// TIA Portal project "2022.11.20_三轴机械臂仿真" (V17)
// Vorlageprojekt für das Buch mit Zielsystem S7-1200

(* hardware
DEVICE "S7-1200-Station_1"  S7-1200 Station
   slot 0: "Baugruppenträger_0"  Rack  V1.0
   slot 1: "PLC_1"  CPU 1214C DC/DC/DC  6ES7 214-1AG40-0XB0  V4.5
*)

// ===== PLC "PLC_1"  CPU 1214C DC/DC/DC =====

VAR_GLOBAL   // PLC tag table "Standard-Variablentabelle"
   "传送带1" AT %A0.0 : Bool;
   "感应器1" AT %E0.0 : Bool;
   "感应器2" AT %E0.1 : Bool;
   "启动" AT %M10.0 : Bool;
   "暂停按钮" AT %I0.2 : Bool;
   "吸物" AT %Q0.3 : Bool;
   "传送带2" AT %Q0.1 : Bool;
   "传送带3" AT %Q0.2 : Bool;
   "上升沿暂存位1" AT %M100.0 : Bool;
   "传送带1输出" AT %M20.0 : Bool;
   "完成" AT %M30.7 : Bool;
   "上升沿暂存位2" AT %M100.1 : Bool;
   "碰上感应1" AT %M30.0 : Bool;
   "传送带3输出" AT %M20.2 : Bool;
   "上升沿暂存位3" AT %M100.2 : Bool;
   "开始拿物" AT %M30.2 : Bool;
   "循环" AT %M30.6 : Bool;
   "碰上感应2" AT %M30.1 : Bool;
   "完成拿物" AT %M30.3 : Bool;
   "X输出" AT %QD30 : Real;
   "Y输出" AT %QD34 : Real;
   "X位置" AT %ID30 : DWord;
   "Y位置" AT %ID34 : DWord;
   "Z输出" AT %QD38 : Real;
   "Z位置" AT %ID38 : DWord;
   "吸物输出" AT %M20.3 : Bool;
   "上升沿暂存位4" AT %M100.3 : Bool;
   "物体个数" AT %MD50 : DWord;
   "X设置输出" AT %MD54 : DWord;
   "Y设置输出" AT %MD58 : DWord;
   "上升沿暂存位5" AT %M100.4 : Bool;
   "X位置(1)" AT %MD62 : Real;
   "Y位置(1)" AT %MD66 : Real;
   "Tag_2" AT %MD34 : DWord;
   "下降" AT %M30.4 : Bool;
   "上升沿暂存位" AT %M100.5 : Bool;
   "Z设置输出" AT %MD70 : Real;
   "Z位置(1)" AT %MD74 : Real;
   "Z位置(2)" AT %MD38 : DWord;
   "上升" AT %M30.5 : Bool;
   "上升沿暂存位(1)" AT %M100.6 : Bool;
   "停止" AT %M10.1 : Bool;
   "Tag_3" AT %M20.1 : Bool;
END_VAR

DATA_BLOCK "拿物_DB"   // DB1
{ S7_Optimized_Access := 'TRUE' }
VERSION : 0.1
// stored: InstanceOfName 拿物
"拿物"
BEGIN
END_DATA_BLOCK

DATA_BLOCK "放物_DB"   // DB10
{ S7_Optimized_Access := 'TRUE' }
VERSION : 0.1
// stored: InstanceOfName 放物
"放物"
BEGIN
END_DATA_BLOCK

DATA_BLOCK "输出_DB"   // DB11
{ S7_Optimized_Access := 'TRUE' }
VERSION : 0.1
// stored: InstanceOfName 输出
"输出"
BEGIN
END_DATA_BLOCK

// folder: System blocks/Program resources

DATA_BLOCK "计数器1"   // DB2
{ S7_Optimized_Access := 'TRUE' }
AUTHOR : Simatic
FAMILY : IEC
NAME : CNTR
VERSION : 1.0
// stored: InstanceOfName IEC_COUNTER
"IEC_COUNTER"
BEGIN
END_DATA_BLOCK

DATA_BLOCK "计数器2"   // DB4
{ S7_Optimized_Access := 'TRUE' }
AUTHOR : Simatic
FAMILY : IEC
NAME : CNTR
VERSION : 1.0
// stored: InstanceOfName IEC_COUNTER
"IEC_COUNTER"
BEGIN
END_DATA_BLOCK

DATA_BLOCK "计时器1"   // DB5
{ S7_Optimized_Access := 'TRUE' }
AUTHOR : Simatic
FAMILY : IEC
NAME : IEC_TMR
VERSION : 1.0
// stored: InstanceOfName IEC_TIMER
"IEC_TIMER"
BEGIN
END_DATA_BLOCK

DATA_BLOCK "计数器3"   // DB6
{ S7_Optimized_Access := 'TRUE' }
AUTHOR : Simatic
FAMILY : IEC
NAME : CNTR
VERSION : 1.0
// stored: InstanceOfName IEC_COUNTER
"IEC_COUNTER"
BEGIN
END_DATA_BLOCK

DATA_BLOCK "计时器2"   // DB7
{ S7_Optimized_Access := 'TRUE' }
AUTHOR : Simatic
FAMILY : IEC
NAME : IEC_TMR
VERSION : 1.0
// stored: InstanceOfName IEC_TIMER
"IEC_TIMER"
BEGIN
END_DATA_BLOCK

DATA_BLOCK "计时2"   // DB8
{ S7_Optimized_Access := 'TRUE' }
AUTHOR : Simatic
FAMILY : IEC
NAME : IEC_TMR
VERSION : 1.0
// stored: InstanceOfName IEC_TIMER
"IEC_TIMER"
BEGIN
END_DATA_BLOCK

DATA_BLOCK "计时1"   // DB9
{ S7_Optimized_Access := 'TRUE' }
AUTHOR : Simatic
FAMILY : IEC
NAME : IEC_TMR
VERSION : 1.0
// stored: InstanceOfName IEC_TIMER
"IEC_TIMER"
BEGIN
END_DATA_BLOCK

// folder: (top level)

FUNCTION_BLOCK "拿物"   // FB1, LAD
{ S7_Optimized_Access := 'TRUE' }
VERSION : 0.1
   VAR_TEMP   // added for the SCL form of the ladder/FBD networks
      _w1 : Bool;
   END_VAR
BEGIN

REGION Network 1: 2个感应碰上后开始拿物
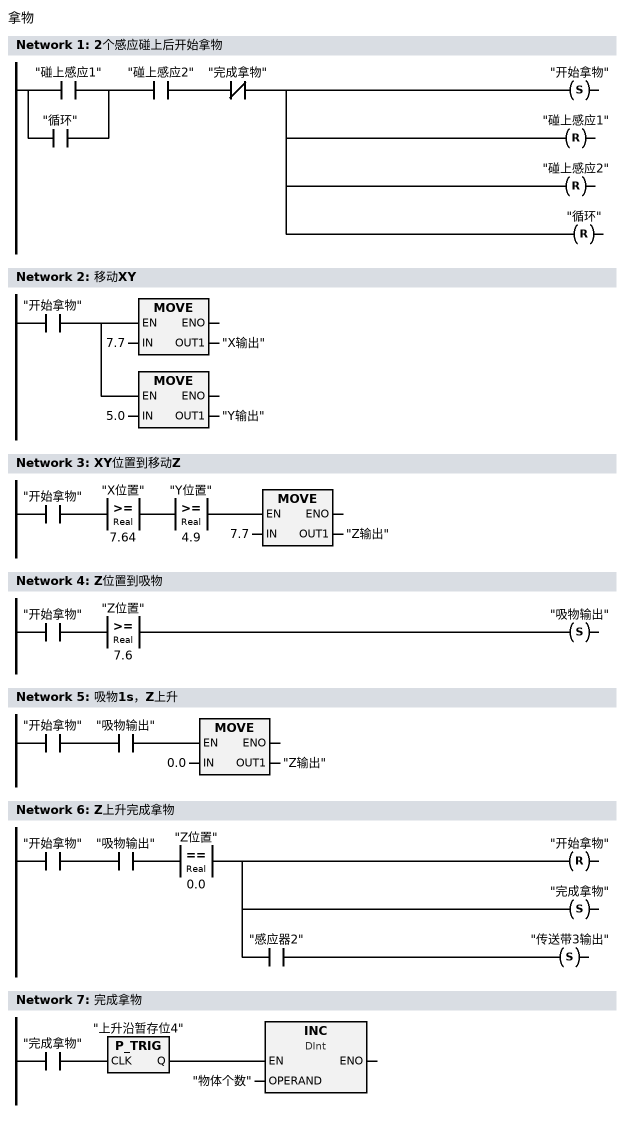
   RUNG wire#powerrail
      Contact( "碰上感应1" )
      wire#w1
      Contact( "碰上感应2" )
      I_Contact( "完成拿物" )
      wire#w2
      S_Coil( "开始拿物" )
   END_RUNG
   RUNG wire#powerrail
      Contact( "循环" )
   END_RUNG wire#w1
   RUNG wire#w2
      R_Coil( "碰上感应1" )
   END_RUNG
   RUNG wire#w2
      R_Coil( "碰上感应2" )
   END_RUNG
   RUNG wire#w2
      R_Coil( "循环" )
   END_RUNG
   // the same network as SCL:
   IF ("碰上感应1" OR "循环") AND "碰上感应2" AND NOT "完成拿物" THEN "开始拿物" := TRUE; END_IF;
   #_w1 := ("碰上感应1" OR "循环") AND "碰上感应2" AND NOT "完成拿物";
   IF #_w1 THEN
       "碰上感应1" := FALSE;
       "碰上感应2" := FALSE;
       "循环" := FALSE;
   END_IF;
END_REGION

REGION Network 2: 移动XY
   RUNG wire#powerrail
      Contact( "开始拿物" )
      wire#w1
      Move(in := 7.7, out1 => "X输出")
   END_RUNG
   RUNG wire#w1
      Move(in := 5.0, out1 => "Y输出")
   END_RUNG
   // the same network as SCL:
   IF "开始拿物" THEN
       "X输出" := 7.7;
       "Y输出" := 5.0;
   END_IF;
END_REGION

REGION Network 3: XY位置到移动Z
   RUNG wire#powerrail
      Contact( "开始拿物" )
      { S7_Templates := "SrcType := Real" } GE_Contact(in1 := "X位置", in2 := 7.64)
      { S7_Templates := "SrcType := Real" } GE_Contact(in1 := "Y位置", in2 := 4.9)
      Move(in := 7.7, out1 => "Z输出")
   END_RUNG
   // the same network as SCL:
   IF "开始拿物" AND ("X位置" >= 7.64) AND ("Y位置" >= 4.9) THEN "Z输出" := 7.7; END_IF;
END_REGION

REGION Network 4: Z位置到吸物
   RUNG wire#powerrail
      Contact( "开始拿物" )
      { S7_Templates := "SrcType := Real" } GE_Contact(in1 := "Z位置", in2 := 7.6)
      S_Coil( "吸物输出" )
   END_RUNG
   // the same network as SCL:
   IF "开始拿物" AND ("Z位置" >= 7.6) THEN "吸物输出" := TRUE; END_IF;
END_REGION

REGION Network 5: 吸物1s，Z上升
   RUNG wire#powerrail
      Contact( "开始拿物" )
      Contact( "吸物输出" )
      Move(in := 0.0, out1 => "Z输出")
   END_RUNG
   // the same network as SCL:
   IF "开始拿物" AND "吸物输出" THEN "Z输出" := 0.0; END_IF;
END_REGION

REGION Network 6: Z上升完成拿物
   RUNG wire#powerrail
      Contact( "开始拿物" )
      Contact( "吸物输出" )
      { S7_Templates := "SrcType := Real" } EQ_Contact(in1 := "Z位置", in2 := 0.0)
      wire#w1
      R_Coil( "开始拿物" )
   END_RUNG
   RUNG wire#w1
      S_Coil( "完成拿物" )
   END_RUNG
   RUNG wire#w1
      Contact( "感应器2" )
      S_Coil( "传送带3输出" )
   END_RUNG
   // the same network as SCL:
   #_w1 := "开始拿物" AND "吸物输出" AND ("Z位置" = 0.0);
   IF #_w1 THEN
       "开始拿物" := FALSE;
       "完成拿物" := TRUE;
   END_IF;
   IF #_w1 AND "感应器2" THEN "传送带3输出" := TRUE; END_IF;
END_REGION

REGION Network 7: 完成拿物
   RUNG wire#powerrail
      Contact( "完成拿物" )
      P_Trig( "上升沿暂存位4" )
      { S7_Templates := "DestType := DInt" } Inc( "物体个数" )
   END_RUNG
   // the same network as SCL:
   #_w1 := "完成拿物" AND NOT "上升沿暂存位4";   // rising edge
   "上升沿暂存位4" := "完成拿物";
   IF #_w1 THEN "物体个数" := "物体个数" + 1; END_IF;
END_REGION
END_FUNCTION_BLOCK

FUNCTION_BLOCK "输出"   // FB2, LAD
{ S7_Optimized_Access := 'TRUE' }
VERSION : 0.1
BEGIN

REGION Network 1
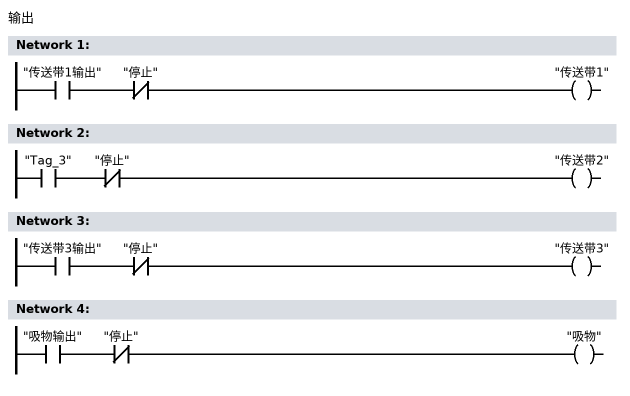
   RUNG wire#powerrail
      Contact( "传送带1输出" )
      I_Contact( "停止" )
      Coil( "传送带1" )
   END_RUNG
   // the same network as SCL:
   "传送带1" := "传送带1输出" AND NOT "停止";
END_REGION

REGION Network 2
   RUNG wire#powerrail
      Contact( "Tag_3" )
      I_Contact( "停止" )
      Coil( "传送带2" )
   END_RUNG
   // the same network as SCL:
   "传送带2" := "Tag_3" AND NOT "停止";
END_REGION

REGION Network 3
   RUNG wire#powerrail
      Contact( "传送带3输出" )
      I_Contact( "停止" )
      Coil( "传送带3" )
   END_RUNG
   // the same network as SCL:
   "传送带3" := "传送带3输出" AND NOT "停止";
END_REGION

REGION Network 4
   RUNG wire#powerrail
      Contact( "吸物输出" )
      I_Contact( "停止" )
      Coil( "吸物" )
   END_RUNG
   // the same network as SCL:
   "吸物" := "吸物输出" AND NOT "停止";
END_REGION
END_FUNCTION_BLOCK

FUNCTION_BLOCK "放物"   // FB3, LAD
{ S7_Optimized_Access := 'TRUE' }
VERSION : 0.1
   VAR_TEMP   // added for the SCL form of the ladder/FBD networks
      _w1 : Bool;
      _w2 : Bool;
   END_VAR
BEGIN

REGION Network 1: Y计数
   // 1. X: 2.3    Y:8.1   2.  X: 4.2   Y:8.0
   // 3. X: 2.3    Y:6.1   4.  X: 4.2   Y:6.0
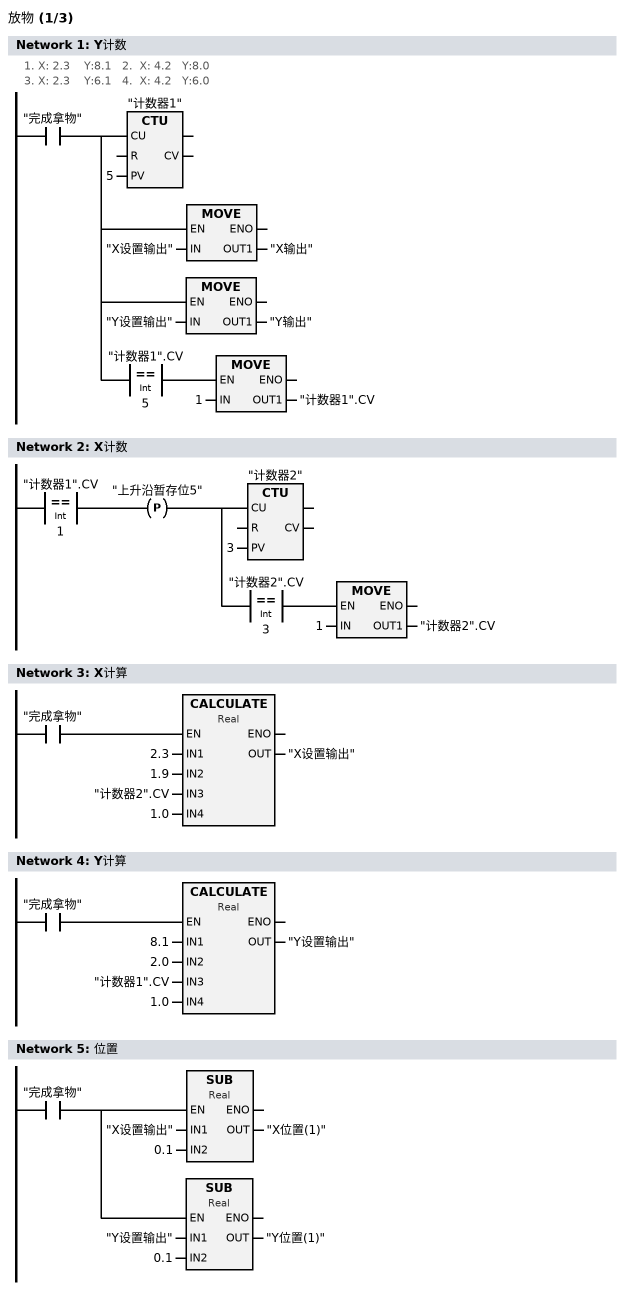
   "计数器1".CTU(CU := "完成拿物", PV := 5);
   IF "完成拿物" THEN
       "X输出" := "X设置输出";
       "Y输出" := "Y设置输出";
   END_IF;
   IF "完成拿物" AND ("计数器1".CV = 5) THEN "计数器1".CV := 1; END_IF;
END_REGION

REGION Network 2: X计数
   #_w1 := "计数器1".CV = 1;
   #_w2 := #_w1 AND NOT "上升沿暂存位5";   // rising edge
   "上升沿暂存位5" := #_w1;
   "计数器2".CTU(CU := #_w2, PV := 3);
   IF #_w2 AND ("计数器2".CV = 3) THEN "计数器2".CV := 1; END_IF;
END_REGION

REGION Network 3: X计算
   RUNG wire#powerrail
      Contact( "完成拿物" )
      { S7_Templates := "SrcType := Real"; S7_Expression := "IN1+IN2*(IN3-IN4)" } Calculate(in1 := 2.3, in2 := 1.9, in3 := "计数器2".CV, in4 := 1.0, out => "X设置输出")
   END_RUNG
   // the same network as SCL:
   IF "完成拿物" THEN "X设置输出" := 2.3+1.9*("计数器2".CV-1.0); END_IF;
END_REGION

REGION Network 4: Y计算
   RUNG wire#powerrail
      Contact( "完成拿物" )
      { S7_Templates := "SrcType := Real"; S7_Expression := "IN1-IN2*(IN3-IN4)" } Calculate(in1 := 8.1, in2 := 2.0, in3 := "计数器1".CV, in4 := 1.0, out => "Y设置输出")
   END_RUNG
   // the same network as SCL:
   IF "完成拿物" THEN "Y设置输出" := 8.1-2.0*("计数器1".CV-1.0); END_IF;
END_REGION

REGION Network 5: 位置
   RUNG wire#powerrail
      Contact( "完成拿物" )
      wire#w1
      { S7_Templates := "SrcType := Real" } Sub(in1 := "X设置输出", in2 := 0.1, out => "X位置(1)")
   END_RUNG
   RUNG wire#w1
      { S7_Templates := "SrcType := Real" } Sub(in1 := "Y设置输出", in2 := 0.1, out => "Y位置(1)")
   END_RUNG
   // the same network as SCL:
   IF "完成拿物" THEN
       "X位置(1)" := "X设置输出" - 0.1;
       "Y位置(1)" := "Y设置输出" - 0.1;
   END_IF;
END_REGION

REGION Network 6: 位置到下降
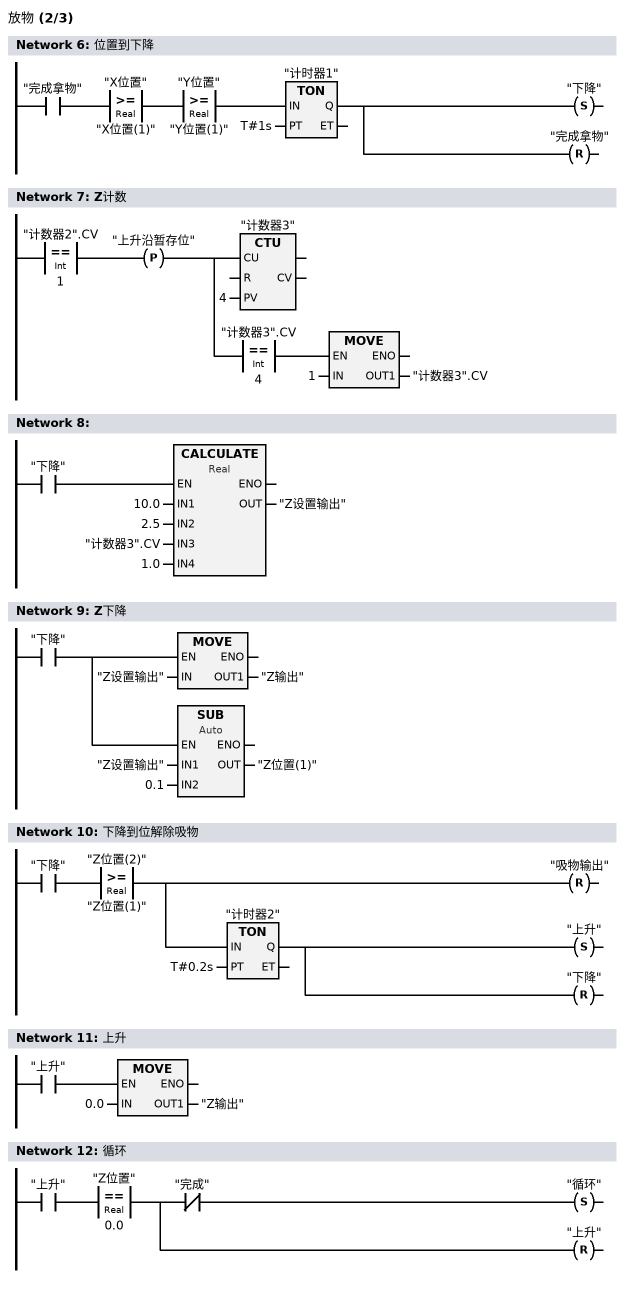
   "计时器1".TON(IN := "完成拿物" AND ("X位置" >= "X位置(1)") AND ("Y位置" >= "Y位置(1)"), PT := T#1s);
   IF "计时器1".Q THEN
       "下降" := TRUE;
       "完成拿物" := FALSE;
   END_IF;
END_REGION

REGION Network 7: Z计数
   #_w1 := "计数器2".CV = 1;
   #_w2 := #_w1 AND NOT "上升沿暂存位";   // rising edge
   "上升沿暂存位" := #_w1;
   "计数器3".CTU(CU := #_w2, PV := 4);
   IF #_w2 AND ("计数器3".CV = 4) THEN "计数器3".CV := 1; END_IF;
END_REGION

REGION Network 8
   RUNG wire#powerrail
      Contact( "下降" )
      { S7_Templates := "SrcType := Real"; S7_Expression := "IN1-IN2*(IN3-IN4)" } Calculate(in1 := 10.0, in2 := 2.5, in3 := "计数器3".CV, in4 := 1.0, out => "Z设置输出")
   END_RUNG
   // the same network as SCL:
   IF "下降" THEN "Z设置输出" := 10.0-2.5*("计数器3".CV-1.0); END_IF;
END_REGION

REGION Network 9: Z下降
   RUNG wire#powerrail
      Contact( "下降" )
      wire#w1
      Move(in := "Z设置输出", out1 => "Z输出")
   END_RUNG
   RUNG wire#w1
      Sub(in1 := "Z设置输出", in2 := 0.1, out => "Z位置(1)")
   END_RUNG
   // the same network as SCL:
   IF "下降" THEN
       "Z输出" := "Z设置输出";
       "Z位置(1)" := "Z设置输出" - 0.1;
   END_IF;
END_REGION

REGION Network 10: 下降到位解除吸物
   #_w1 := "下降" AND ("Z位置(2)" >= "Z位置(1)");
   IF #_w1 THEN "吸物输出" := FALSE; END_IF;
   "计时器2".TON(IN := #_w1, PT := T#0.2s);
   IF "计时器2".Q THEN
       "上升" := TRUE;
       "下降" := FALSE;
   END_IF;
END_REGION

REGION Network 11: 上升
   RUNG wire#powerrail
      Contact( "上升" )
      Move(in := 0.0, out1 => "Z输出")
   END_RUNG
   // the same network as SCL:
   IF "上升" THEN "Z输出" := 0.0; END_IF;
END_REGION

REGION Network 12: 循环
   RUNG wire#powerrail
      Contact( "上升" )
      { S7_Templates := "SrcType := Real" } EQ_Contact(in1 := "Z位置", in2 := 0.0)
      wire#w1
      I_Contact( "完成" )
      S_Coil( "循环" )
   END_RUNG
   RUNG wire#w1
      R_Coil( "上升" )
   END_RUNG
   // the same network as SCL:
   #_w1 := "上升" AND ("Z位置" = 0.0);
   IF #_w1 AND NOT "完成" THEN "循环" := TRUE; END_IF;
   IF #_w1 THEN "上升" := FALSE; END_IF;
END_REGION

REGION Network 13: 完成
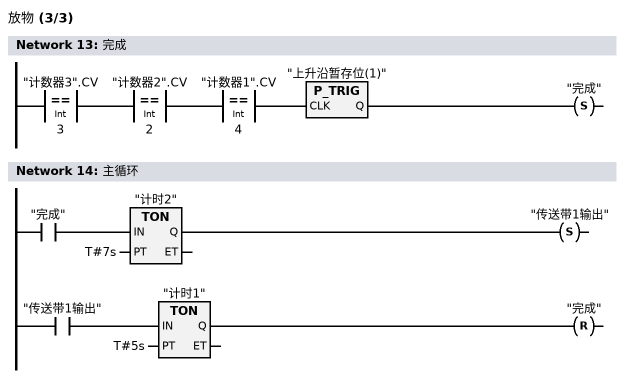
   RUNG wire#powerrail
      { S7_Templates := "SrcType := Int" } EQ_Contact(in1 := "计数器3".CV, in2 := 3)
      { S7_Templates := "SrcType := Int" } EQ_Contact(in1 := "计数器2".CV, in2 := 2)
      { S7_Templates := "SrcType := Int" } EQ_Contact(in1 := "计数器1".CV, in2 := 4)
      P_Trig( "上升沿暂存位(1)" )
      S_Coil( "完成" )
   END_RUNG
   // the same network as SCL:
   #_w1 := ("计数器3".CV = 3) AND ("计数器2".CV = 2) AND ("计数器1".CV = 4);
   #_w2 := #_w1 AND NOT "上升沿暂存位(1)";   // rising edge
   "上升沿暂存位(1)" := #_w1;
   IF #_w2 THEN "完成" := TRUE; END_IF;
END_REGION

REGION Network 14: 主循环
   "计时2".TON(IN := "完成", PT := T#7s);
   IF "计时2".Q THEN "传送带1输出" := TRUE; END_IF;
   "计时1".TON(IN := "传送带1输出", PT := T#5s);
   IF "计时1".Q THEN "完成" := FALSE; END_IF;
END_REGION
END_FUNCTION_BLOCK

FUNCTION "MHJ-PLC-Lab-Function-S71200" : Void   // FC9000, SCL
{ S7_Optimized_Access := 'TRUE' }
VERSION : 0.1
   VAR_TEMP
      rdTimeReturn : Int;
      outputTime : DTL;
      SyncVal : Byte;
      forVal : Int;
      forVal_2 : Int;
      Value : Byte;
   END_VAR
   VAR CONSTANT
      CompVal : Byte := 16#34;
      Value_01 : Byte := 16#11;
      Value_01_DW : DWord := 16#A165_D992;
      Value_02_DW : DWord := 16#58BE_4401;
   END_VAR
BEGIN

   #Value:=PEEK(area := 16#82,
        dbNumber := 0,
        byteOffset := 511);
   #Value := #Value + 1;

   POKE(area := 16#82,
        dbNumber := 0,
        byteOffset := 511,
        value := #Value);

   POKE(area:=16#81,
        dbNumber:=0,
        byteOffset:=1016,
        value:=#Value_01_DW);
   POKE(area := 16#81,
        dbNumber := 0,
        byteOffset := 1020,
        value := #Value_02_DW);

   POKE(area := 16#81,
        dbNumber := 0,
        byteOffset := 511,
        value := B#16#00);

   FOR #forVal := 0 TO 120 DO
       FOR #forVal_2:=0 TO 10 DO
           #rdTimeReturn:=RD_SYS_T(#outputTime);
           #rdTimeReturn := WR_SYS_T(#outputTime);
           #rdTimeReturn := RD_SYS_T(#outputTime);
           #rdTimeReturn := WR_SYS_T(#outputTime);
       END_FOR;
       #SyncVal:= PEEK(area := 16#81,
                      dbNumber := 0,
                      byteOffset := 511);
       IF #SyncVal = #CompVal THEN
          GOTO M_1;
       END_IF;
   END_FOR;
   RETURN;

   M_1:
   POKE(area := 16#81,
        dbNumber := 0,
        byteOffset := 511,
        value := B#16#0);
END_FUNCTION

ORGANIZATION_BLOCK "Main"   // OB1, LAD, ProgramCycle
TITLE = "Main Program Sweep (Cycle)"
{ S7_Optimized_Access := 'TRUE' }
VERSION : 0.1
   VAR_INPUT
      Initial_Call : Bool;   // Initial call of this OB
      Remanence : Bool;   // =True, if remanent data are available
   END_VAR
   VAR_TEMP   // added for the SCL form of the ladder/FBD networks
      _w1 : Bool;
      _w2 : Bool;
   END_VAR
BEGIN

REGION Network 1
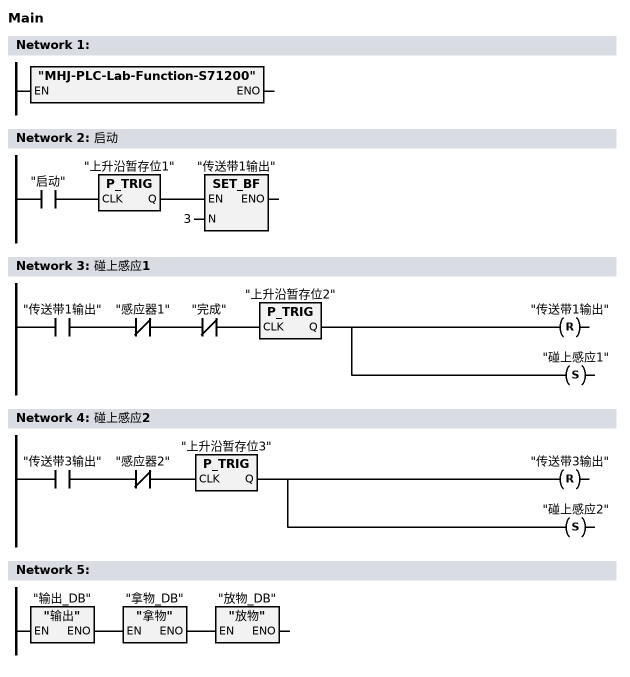
   RUNG wire#powerrail
      "MHJ-PLC-Lab-Function-S71200"()
   END_RUNG
   // the same network as SCL:
   "MHJ-PLC-Lab-Function-S71200"();
END_REGION

REGION Network 2: 启动
   // no SCL statement known for SBitfield: written as a call
   #_w1 := "启动" AND NOT "上升沿暂存位1";   // rising edge
   "上升沿暂存位1" := "启动";
   IF #_w1 THEN SET_BF(operand := "传送带1输出", n := 3); END_IF;
END_REGION

REGION Network 3: 碰上感应1
   RUNG wire#powerrail
      Contact( "传送带1输出" )
      I_Contact( "感应器1" )
      I_Contact( "完成" )
      P_Trig( "上升沿暂存位2" )
      wire#w1
      R_Coil( "传送带1输出" )
   END_RUNG
   RUNG wire#w1
      S_Coil( "碰上感应1" )
   END_RUNG
   // the same network as SCL:
   #_w1 := "传送带1输出" AND NOT "感应器1" AND NOT "完成";
   #_w2 := #_w1 AND NOT "上升沿暂存位2";   // rising edge
   "上升沿暂存位2" := #_w1;
   IF #_w2 THEN
       "传送带1输出" := FALSE;
       "碰上感应1" := TRUE;
   END_IF;
END_REGION

REGION Network 4: 碰上感应2
   RUNG wire#powerrail
      Contact( "传送带3输出" )
      I_Contact( "感应器2" )
      P_Trig( "上升沿暂存位3" )
      wire#w1
      R_Coil( "传送带3输出" )
   END_RUNG
   RUNG wire#w1
      S_Coil( "碰上感应2" )
   END_RUNG
   // the same network as SCL:
   #_w1 := "传送带3输出" AND NOT "感应器2";
   #_w2 := #_w1 AND NOT "上升沿暂存位3";   // rising edge
   "上升沿暂存位3" := #_w1;
   IF #_w2 THEN
       "传送带3输出" := FALSE;
       "碰上感应2" := TRUE;
   END_IF;
END_REGION

REGION Network 5
   RUNG wire#powerrail
      "输出_DB"()
      "拿物_DB"()
      "放物_DB"()
   END_RUNG
   // the same network as SCL:
   "输出_DB"(ENO => #_w1);   // "输出"
   "拿物_DB"(EN := #_w1, ENO => #_w2);   // "拿物"
   IF #_w2 THEN
       "放物_DB"();   // "放物"
   END_IF;
END_REGION
END_ORGANIZATION_BLOCK